FUNCTION F_MbExpectedResponseLength : UINT
VAR_INPUT
	nFc  : USINT;
	nQty : UINT;
END_VAR

// PDU bytes of a normal response (no unit ID, CRC or MBAP). 0 = unsupported FC.
// An exception response is always 2 PDU bytes; transports check for that separately.
CASE nFc OF
	GVL_MbConst.FC_READ_COILS, GVL_MbConst.FC_READ_DISCRETE:
		F_MbExpectedResponseLength := 2 + (nQty + 7) / 8;
	GVL_MbConst.FC_READ_HOLDING, GVL_MbConst.FC_READ_INPUT:
		F_MbExpectedResponseLength := 2 + 2 * nQty;
	GVL_MbConst.FC_WRITE_COIL, GVL_MbConst.FC_WRITE_REGISTER,
	GVL_MbConst.FC_WRITE_COILS, GVL_MbConst.FC_WRITE_REGISTERS:
		F_MbExpectedResponseLength := 5;
ELSE
	F_MbExpectedResponseLength := 0;
END_CASE

END_FUNCTION

(* stored: Version 1.1.0.1
   POU F_MbExpectedResponseLength: Id {e2337f90-aa96-4802-8191-50ceeac9ead2}, SpecialFunc None *)
